(* Schneider Machine Expert - Basic project GreenFeed_Lift_TM100, file version 1.5.0.0 *)
(* ProjectInformations: Name=New project *)

HARDWARE
  Cpu 0: TM100C24R
  EthernetConfiguration: NetworkName=M221, IpAllocationMode=FixedAddress, IpAddress=0.0.0.0, SubnetMask=0.0.0.0
  SerialLineConfiguration: Baud=Baud19200, Parity=ParityEven, DataBits=DataBits8, StopBits=StopBits1, PhysicalMedium=PhysicalMediumRs485, TransmissionMode=TransmissionModeModbusRtu, SlaveId=1, Addressing=SlaveAddressing
  MastTask: UsePeriodScanMode=false, PeriodScan=100
  FastTask: Period=255
  CpuBehavior: StartingMode=StartAsPreviousState, AutoSaveRamOnEeprom=true, WatchdogPeriod=250

SYMBOLS  (address, symbol, comment, settings)
  %M0       GOTOFLOOR2
  %M1       MOVEUP
  %M2       MOVEDOWN
  %M3       GOTOFLOOR1
  %M4       GODOWN
  %M5       GOUP
  %M6       GOTOFLOOR3
  %M7       GOUP2
  %M8       GODOWN2
  %M9       MOVEUP2
  %M10      MOVEDOWN2
  %M11      GOTOFLOOR4
  %I0.0     ESTOP
  %I0.1     BOTTOMLS
  %I0.2     TOPLS
  %I0.3     FLOOR1LS
  %I0.4     FLOOR2LS
  %I0.5     FLOOR3LS
  %I0.6     FLOOR1PB
  %I0.7     FLOOR2PB
  %I0.8     FLOOR3PB
  %I0.9     FLOOR4LS
  %I0.10    FLOOR4PB
  %Q0.0     UPCMD
  %Q0.1     DOWNCMD
  %Q0.2     FLOOR1IND
  %Q0.3     FLOOR2IND
  %Q0.4     FLOOR3IND
  %Q0.5     FLOOR4IND

POU New POU
  (* SectionNumber=1, IsGrafcet=false *)

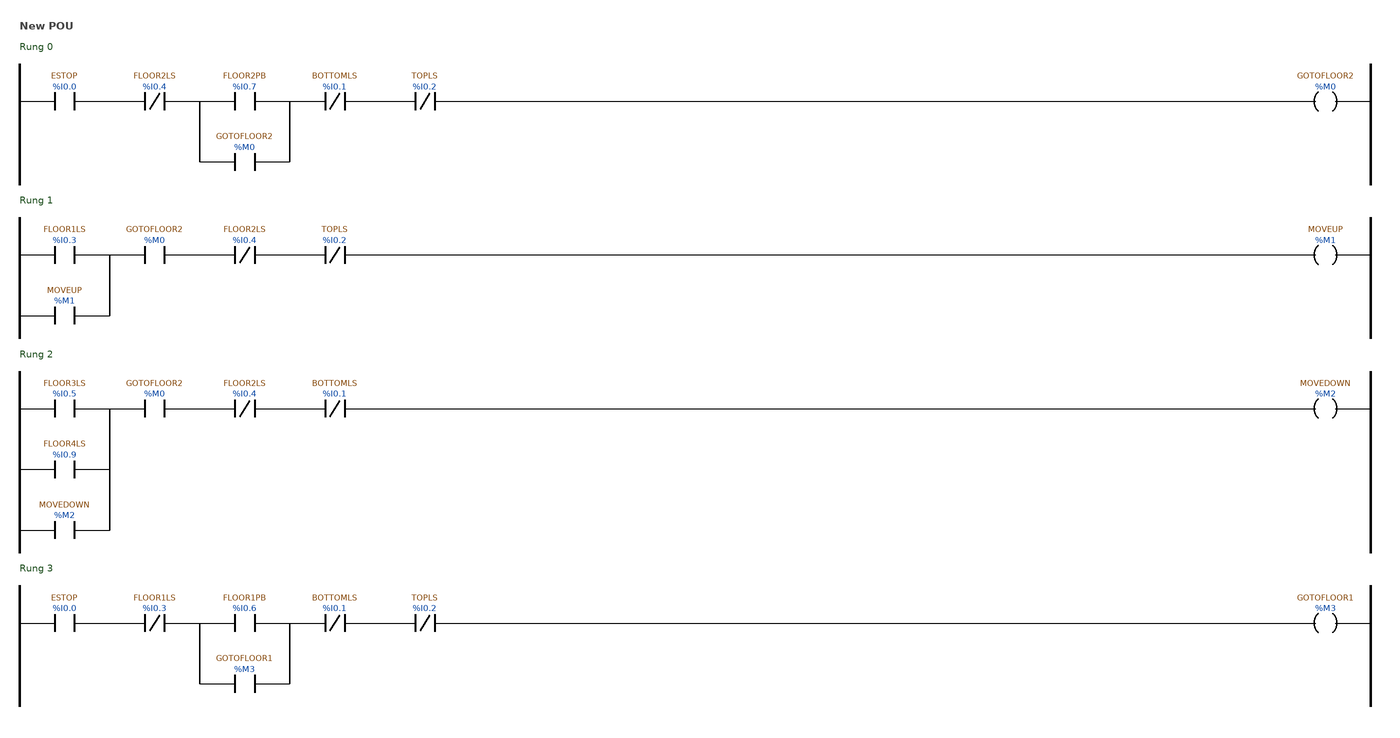

// Rung 0
  LD %I0.0                (* ESTOP *)
  ANDN %I0.4              (* FLOOR2LS *)
  AND( %I0.7              (* FLOOR2PB *)
  OR %M0                  (* GOTOFLOOR2 *)
  )
  ANDN %I0.1              (* BOTTOMLS *)
  ANDN %I0.2              (* TOPLS *)
  ST %M0                  (* GOTOFLOOR2 *)
  // as ST:
  //   GOTOFLOOR2 := ESTOP AND NOT FLOOR2LS AND (FLOOR2PB OR GOTOFLOOR2) AND NOT BOTTOMLS AND NOT TOPLS;

// Rung 1
  LD %I0.3                (* FLOOR1LS *)
  OR %M1                  (* MOVEUP *)
  AND %M0                 (* GOTOFLOOR2 *)
  ANDN %I0.4              (* FLOOR2LS *)
  ANDN %I0.2              (* TOPLS *)
  ST %M1                  (* MOVEUP *)
  // as ST:
  //   MOVEUP := (FLOOR1LS OR MOVEUP) AND GOTOFLOOR2 AND NOT FLOOR2LS AND NOT TOPLS;

// Rung 2
  LD %I0.5                (* FLOOR3LS *)
  OR %I0.9                (* FLOOR4LS *)
  OR %M2                  (* MOVEDOWN *)
  AND %M0                 (* GOTOFLOOR2 *)
  ANDN %I0.4              (* FLOOR2LS *)
  ANDN %I0.1              (* BOTTOMLS *)
  ST %M2                  (* MOVEDOWN *)
  // as ST:
  //   MOVEDOWN := (FLOOR3LS OR FLOOR4LS OR MOVEDOWN) AND GOTOFLOOR2 AND NOT FLOOR2LS AND NOT BOTTOMLS;

// Rung 3
  LD %I0.0                (* ESTOP *)
  ANDN %I0.3              (* FLOOR1LS *)
  AND( %I0.6              (* FLOOR1PB *)
  OR %M3                  (* GOTOFLOOR1 *)
  )
  ANDN %I0.1              (* BOTTOMLS *)
  ANDN %I0.2              (* TOPLS *)
  ST %M3                  (* GOTOFLOOR1 *)
  // as ST:
  //   GOTOFLOOR1 := ESTOP AND NOT FLOOR1LS AND (FLOOR1PB OR GOTOFLOOR1) AND NOT BOTTOMLS AND NOT TOPLS;

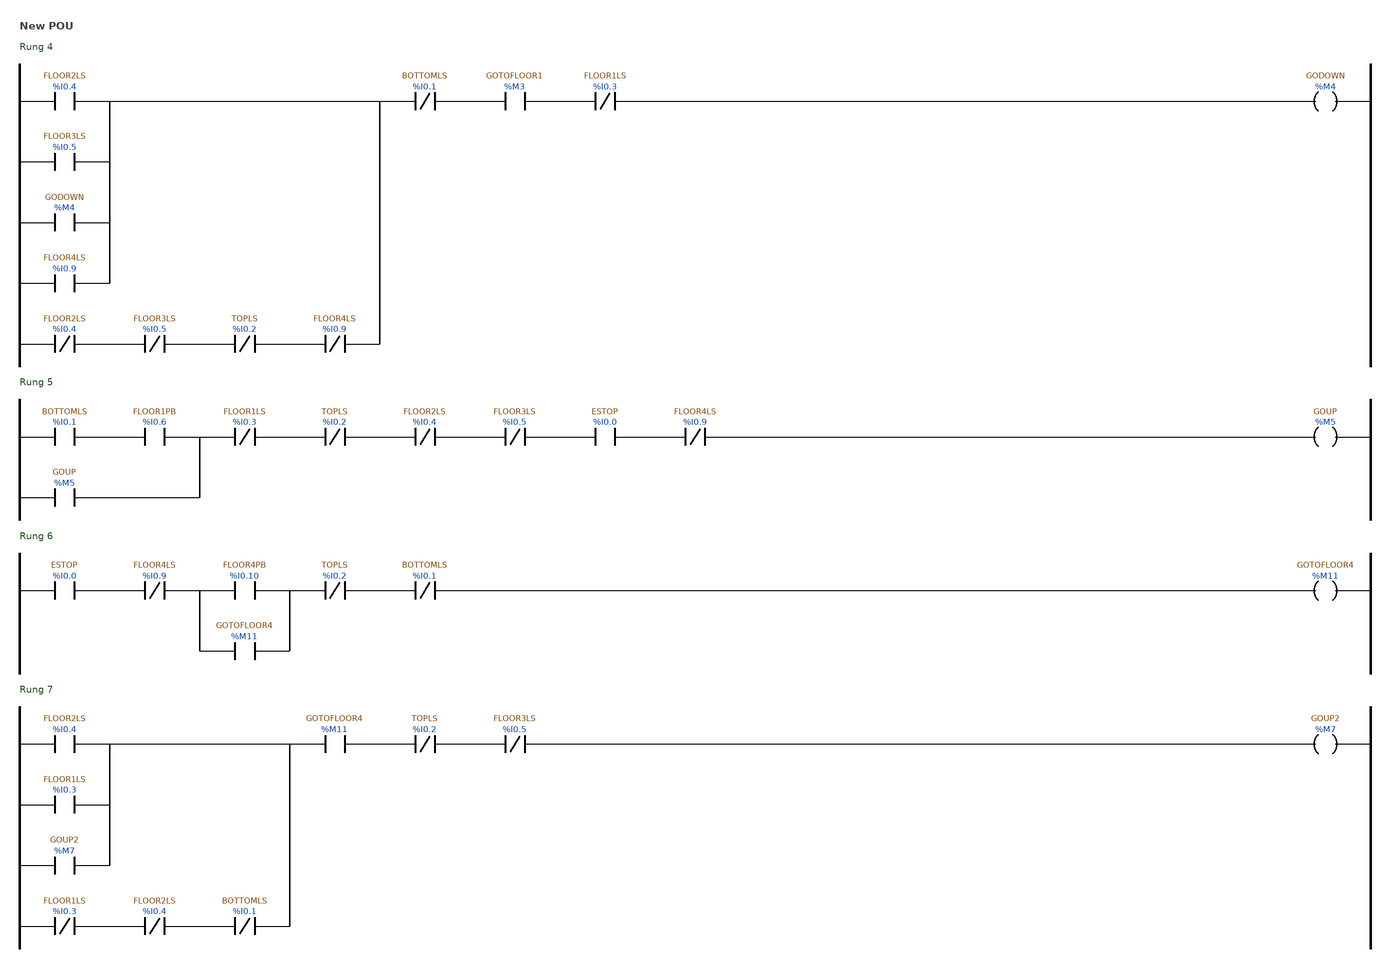

// Rung 4
  LD %I0.4                (* FLOOR2LS *)
  OR %I0.5                (* FLOOR3LS *)
  OR %M4                  (* GODOWN *)
  OR %I0.9                (* FLOOR4LS *)
  OR(N %I0.4              (* FLOOR2LS *)
  ANDN %I0.5              (* FLOOR3LS *)
  ANDN %I0.2              (* TOPLS *)
  ANDN %I0.9              (* FLOOR4LS *)
  )
  ANDN %I0.1              (* BOTTOMLS *)
  AND %M3                 (* GOTOFLOOR1 *)
  ANDN %I0.3              (* FLOOR1LS *)
  ST %M4                  (* GODOWN *)
  // as ST:
  //   GODOWN := (FLOOR2LS OR FLOOR3LS OR GODOWN OR FLOOR4LS OR NOT FLOOR2LS AND NOT FLOOR3LS AND NOT TOPLS AND NOT FLOOR4LS) AND NOT BOTTOMLS AND GOTOFLOOR1 AND NOT FLOOR1LS;

// Rung 5
  LD %I0.1                (* BOTTOMLS *)
  AND %I0.6               (* FLOOR1PB *)
  OR %M5                  (* GOUP *)
  ANDN %I0.3              (* FLOOR1LS *)
  ANDN %I0.2              (* TOPLS *)
  ANDN %I0.4              (* FLOOR2LS *)
  ANDN %I0.5              (* FLOOR3LS *)
  AND %I0.0               (* ESTOP *)
  ANDN %I0.9              (* FLOOR4LS *)
  ST %M5                  (* GOUP *)
  // as ST:
  //   GOUP := (BOTTOMLS AND FLOOR1PB OR GOUP) AND NOT FLOOR1LS AND NOT TOPLS AND NOT FLOOR2LS AND NOT FLOOR3LS AND ESTOP AND NOT FLOOR4LS;

// Rung 6
  LD %I0.0                (* ESTOP *)
  ANDN %I0.9              (* FLOOR4LS *)
  AND( %I0.10             (* FLOOR4PB *)
  OR %M11                 (* GOTOFLOOR4 *)
  )
  ANDN %I0.2              (* TOPLS *)
  ANDN %I0.1              (* BOTTOMLS *)
  ST %M11                 (* GOTOFLOOR4 *)
  // as ST:
  //   GOTOFLOOR4 := ESTOP AND NOT FLOOR4LS AND (FLOOR4PB OR GOTOFLOOR4) AND NOT TOPLS AND NOT BOTTOMLS;

// Rung 7
  LD %I0.4                (* FLOOR2LS *)
  OR %I0.3                (* FLOOR1LS *)
  OR %M7                  (* GOUP2 *)
  OR(N %I0.3              (* FLOOR1LS *)
  ANDN %I0.4              (* FLOOR2LS *)
  ANDN %I0.1              (* BOTTOMLS *)
  )
  AND %M11                (* GOTOFLOOR4 *)
  ANDN %I0.2              (* TOPLS *)
  ANDN %I0.5              (* FLOOR3LS *)
  ST %M7                  (* GOUP2 *)
  // as ST:
  //   GOUP2 := (FLOOR2LS OR FLOOR1LS OR GOUP2 OR NOT FLOOR1LS AND NOT FLOOR2LS AND NOT BOTTOMLS) AND GOTOFLOOR4 AND NOT TOPLS AND NOT FLOOR3LS;

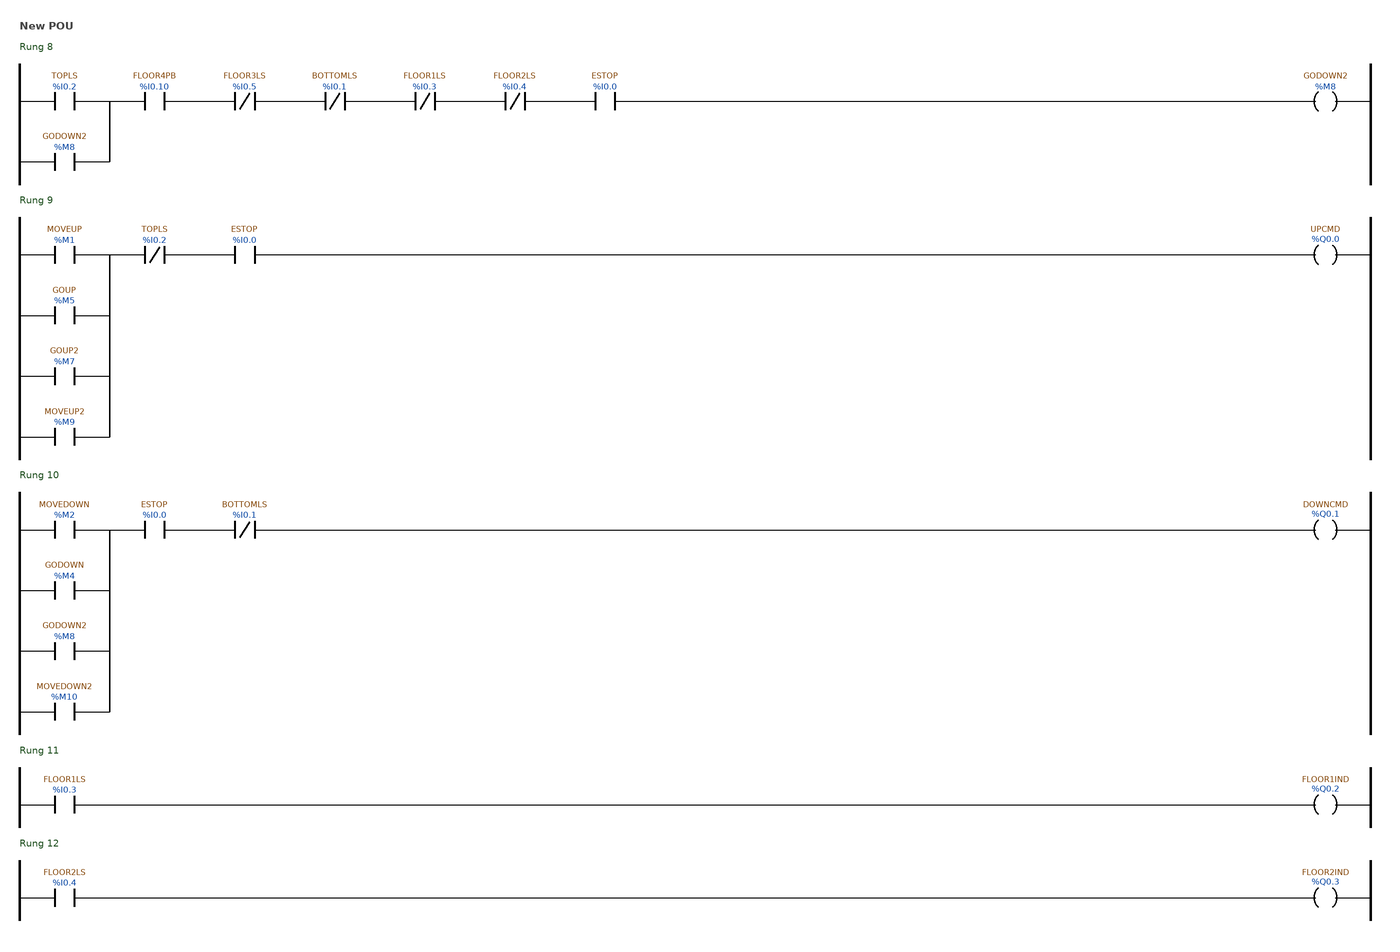

// Rung 8
  LD %I0.2                (* TOPLS *)
  OR %M8                  (* GODOWN2 *)
  AND %I0.10              (* FLOOR4PB *)
  ANDN %I0.5              (* FLOOR3LS *)
  ANDN %I0.1              (* BOTTOMLS *)
  ANDN %I0.3              (* FLOOR1LS *)
  ANDN %I0.4              (* FLOOR2LS *)
  AND %I0.0               (* ESTOP *)
  ST %M8                  (* GODOWN2 *)
  // as ST:
  //   GODOWN2 := (TOPLS OR GODOWN2) AND FLOOR4PB AND NOT FLOOR3LS AND NOT BOTTOMLS AND NOT FLOOR1LS AND NOT FLOOR2LS AND ESTOP;

// Rung 9
  LD %M1                  (* MOVEUP *)
  OR %M5                  (* GOUP *)
  OR %M7                  (* GOUP2 *)
  OR %M9                  (* MOVEUP2 *)
  ANDN %I0.2              (* TOPLS *)
  AND %I0.0               (* ESTOP *)
  ST %Q0.0                (* UPCMD *)
  // as ST:
  //   UPCMD := (MOVEUP OR GOUP OR GOUP2 OR MOVEUP2) AND NOT TOPLS AND ESTOP;

// Rung 10
  LD %M2                  (* MOVEDOWN *)
  OR %M4                  (* GODOWN *)
  OR %M8                  (* GODOWN2 *)
  OR %M10                 (* MOVEDOWN2 *)
  AND %I0.0               (* ESTOP *)
  ANDN %I0.1              (* BOTTOMLS *)
  ST %Q0.1                (* DOWNCMD *)
  // as ST:
  //   DOWNCMD := (MOVEDOWN OR GODOWN OR GODOWN2 OR MOVEDOWN2) AND ESTOP AND NOT BOTTOMLS;

// Rung 11
  LD %I0.3                (* FLOOR1LS *)
  ST %Q0.2                (* FLOOR1IND *)
  // as ST:
  //   FLOOR1IND := FLOOR1LS;

// Rung 12
  LD %I0.4                (* FLOOR2LS *)
  ST %Q0.3                (* FLOOR2IND *)
  // as ST:
  //   FLOOR2IND := FLOOR2LS;

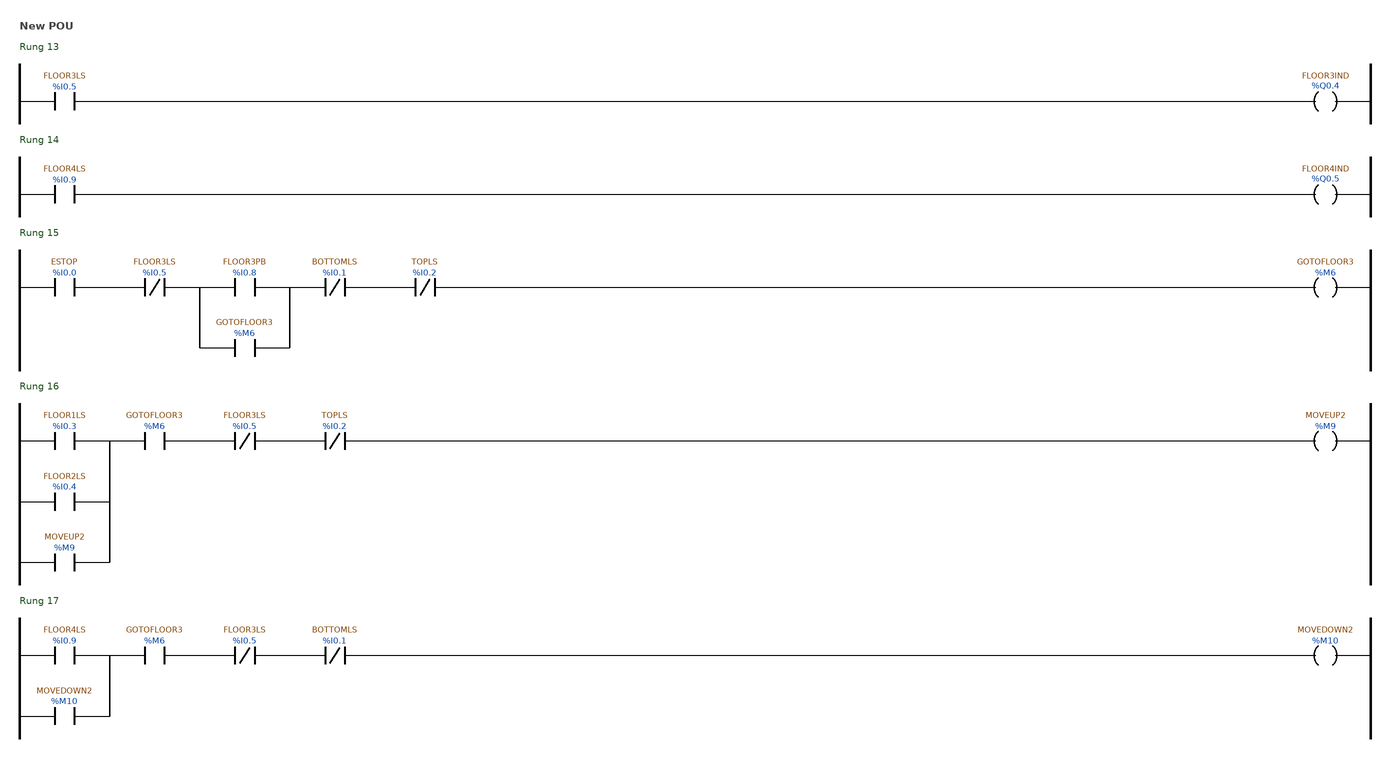

// Rung 13
  LD %I0.5                (* FLOOR3LS *)
  ST %Q0.4                (* FLOOR3IND *)
  // as ST:
  //   FLOOR3IND := FLOOR3LS;

// Rung 14
  LD %I0.9                (* FLOOR4LS *)
  ST %Q0.5                (* FLOOR4IND *)
  // as ST:
  //   FLOOR4IND := FLOOR4LS;

// Rung 15
  LD %I0.0                (* ESTOP *)
  ANDN %I0.5              (* FLOOR3LS *)
  AND( %I0.8              (* FLOOR3PB *)
  OR %M6                  (* GOTOFLOOR3 *)
  )
  ANDN %I0.1              (* BOTTOMLS *)
  ANDN %I0.2              (* TOPLS *)
  ST %M6                  (* GOTOFLOOR3 *)
  // as ST:
  //   GOTOFLOOR3 := ESTOP AND NOT FLOOR3LS AND (FLOOR3PB OR GOTOFLOOR3) AND NOT BOTTOMLS AND NOT TOPLS;

// Rung 16
  LD %I0.3                (* FLOOR1LS *)
  OR %I0.4                (* FLOOR2LS *)
  OR %M9                  (* MOVEUP2 *)
  AND %M6                 (* GOTOFLOOR3 *)
  ANDN %I0.5              (* FLOOR3LS *)
  ANDN %I0.2              (* TOPLS *)
  ST %M9                  (* MOVEUP2 *)
  // as ST:
  //   MOVEUP2 := (FLOOR1LS OR FLOOR2LS OR MOVEUP2) AND GOTOFLOOR3 AND NOT FLOOR3LS AND NOT TOPLS;

// Rung 17
  LD %I0.9                (* FLOOR4LS *)
  OR %M10                 (* MOVEDOWN2 *)
  AND %M6                 (* GOTOFLOOR3 *)
  ANDN %I0.5              (* FLOOR3LS *)
  ANDN %I0.1              (* BOTTOMLS *)
  ST %M10                 (* MOVEDOWN2 *)
  // as ST:
  //   MOVEDOWN2 := (FLOOR4LS OR MOVEDOWN2) AND GOTOFLOOR3 AND NOT FLOOR3LS AND NOT BOTTOMLS;
